{attribute 'GeneratedUsingTerminal: EJ7211-9414-0030'}
{attribute addProperty BoxType "EJ7211-9414-0030"}
{attribute addProperty Description "EJ7211-9414 1Ch. MDP742 Servo motor output stage with OCT (50V, 4.5A RMS) , TwinSAFE SC"}
{attribute addProperty Physics "KK"}
{attribute addProperty Id "FB_PositionAT %I*FB_Position_3FA094ED4DRV_StatuswordAT %I*DRV_Statusword_9B36FDFC2DRV_ControlwordAT %Q*DRV_Controlword_F3F147212DRV_Target_velocityAT %Q*DRV_Target_velocity_08A9583B4WcStateAT %I*WcState_9091E0EB2InfoDataAT %I*InfoData_8300A75E21"}
{attribute addProperty CRC "3086397267"}
{attribute addProperty Size "35"}
TYPE EJ7211_B7F6AF53 EXTENDS EtcSlaveTerminalBase_947E5A46 :
STRUCT
	{attribute addProperty Name "FB_Position"}
	FB_Position : FB_Position_3FA094ED;
	{attribute addProperty Name "DRV_Statusword"}
	DRV_Statusword : DRV_Statusword_9B36FDFC;
	{attribute addProperty Name "DRV_Controlword"}
	DRV_Controlword : DRV_Controlword_F3F14721;
	{attribute addProperty Name "DRV_Target_velocity"}
	DRV_Target_velocity : DRV_Target_velocity_08A9583B;
	{attribute addProperty Name "WcState"}
	WcState : WcState_9091E0EB;
	{attribute addProperty Name "InfoData"}
	InfoData : InfoData_8300A75E;
END_STRUCT
END_TYPE

(* stored: Version 1.2.0.0, ProductVersion 3.1.4024.9
   DUT EJ7211_B7F6AF53: Id {d1243b1f-0ca8-4409-8d40-6563ac44c82b} *)
